{attribute 'GeneratedUsingTerminal: EPP7041-1002-0016'}
{attribute addProperty BoxType "EPP7041-1002-0016"}
{attribute addProperty Description "EPP7041-1002 1Ch. Stepper motor output stage (50V, 1.5A)"}
{attribute addProperty Physics "YY"}
{attribute addProperty Id "ENC_Status_compactAT %I*ENC_Status_compact_4D066E1A16STM_StatusAT %I*STM_Status_36ED096F11ENC_Control_compactAT %Q*ENC_Control_compact_21E2D14D6STM_ControlAT %Q*STM_Control_BA4CE3524STM_VelocityAT %Q*STM_Velocity_A47A3F412WcStateAT %I*WcState_9091E0EB2InfoDataAT %I*InfoData_6538CF5F12"}
{attribute addProperty CRC "839962432"}
{attribute addProperty Size "53"}
TYPE EPP7041_3210CF40 EXTENDS EtcSlaveBoxBase_77A0E4A7 :
STRUCT
	{attribute addProperty Name "ENC_Status_compact"}
	ENC_Status_compact : ENC_Status_compact_4D066E1A;
	{attribute addProperty Name "STM_Status"}
	STM_Status : STM_Status_36ED096F;
	{attribute addProperty Name "ENC_Control_compact"}
	ENC_Control_compact : ENC_Control_compact_21E2D14D;
	{attribute addProperty Name "STM_Control"}
	STM_Control : STM_Control_BA4CE352;
	{attribute addProperty Name "STM_Velocity"}
	STM_Velocity : STM_Velocity_A47A3F41;
	{attribute addProperty Name "WcState"}
	WcState : WcState_9091E0EB;
	{attribute addProperty Name "InfoData"}
	InfoData : InfoData_6538CF5F;
END_STRUCT
END_TYPE

(* stored: Version 1.2.0.0, ProductVersion 3.1.4024.9
   DUT EPP7041_3210CF40: Id {9035cc3e-d223-402f-904c-a6473524a2ff} *)
